INTERFACE I_Axis_PTP EXTENDS I_Axis, I_AxisMoveAbsolute, I_AxisMoveModulo, I_AxisMoveRelative, I_AxisMoveVelocity

END_INTERFACE

(* stored: Version 1.1.0.1, ProductVersion 3.1.4026.18
   Itf I_Axis_PTP: Id {bfe1ba3a-5906-4db0-8de5-4bed3b573cf8} *)
